{attribute 'GeneratedUsingTerminal: IndraDrive MPB20-0003-0000'}
{attribute addProperty BoxType "IndraDrive MPB20-0003-0000"}
{attribute addProperty Id "Drive_status_wordAT %I*UINT2Position_feedback_value_1AT %I*DINT4Following_distanceAT %I*DINT4"}
{attribute addProperty CRC "1197227380"}
{attribute addProperty Size "10"}
TYPE AT_x_475C3D74 EXTENDS TcoIo.InputBase_8311D824 :
STRUCT
	{attribute addProperty Name "Drive_status_word"}
	Drive_status_word AT %I* : UINT;
	{attribute addProperty Name "Position_feedback_value_1"}
	Position_feedback_value_1 AT %I* : DINT;
	{attribute addProperty Name "Following_distance"}
	Following_distance AT %I* : DINT;
END_STRUCT
END_TYPE

(* stored: Version 1.2.0.0, ProductVersion 3.1.4024.9
   DUT AT_x_475C3D74: Id {c888a143-f655-0e3e-0d86-57324226a851} *)
